PROGRAM StartStop
VAR
	Start:BOOL;	
	Stop:BOOL;	
    Run:BOOL;
	PulseOUT:BOOL;
	Value:INT;
	TOn:TON;	
	Rtrig:R_TRIG;
	TOn_ET: TIME;
	FAIZ: BOOL;
	FAIZV: INT;
	FAIZValue1 : INT;
	FAIZValue2 : INT;
END_VAR

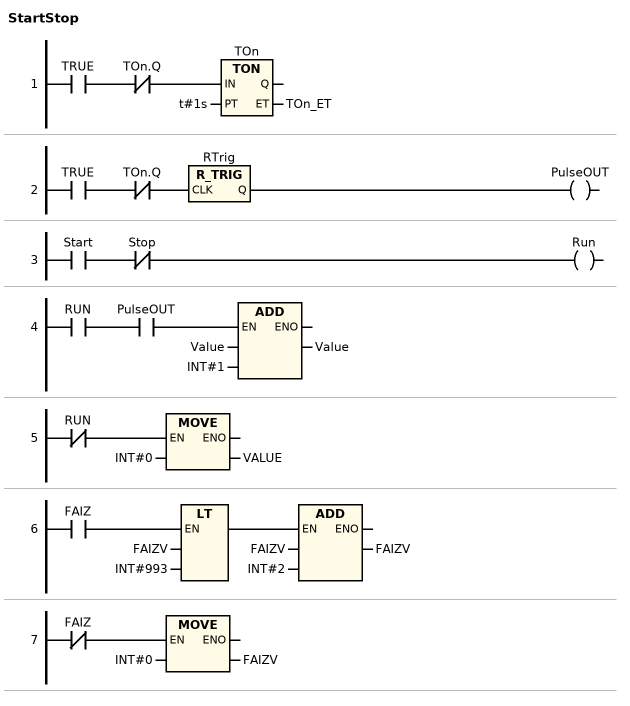
// NETWORK 1
TOn(IN := TRUE AND NOT TOn.Q, PT := t#1s, ET => TOn_ET);

// NETWORK 2
RTrig(CLK := TRUE AND NOT TOn.Q); // R_TRIG
PulseOUT := RTrig.Q;

// NETWORK 3
Run := Start AND NOT Stop;

// NETWORK 4
IF RUN AND PulseOUT THEN Value := Value + INT#1; END_IF

// NETWORK 5
IF NOT RUN THEN VALUE := INT#0; END_IF

// NETWORK 6
IF FAIZ AND FAIZV < INT#993 THEN FAIZV := FAIZV + INT#2; END_IF

// NETWORK 7
IF NOT FAIZ THEN FAIZV := INT#0; END_IF

END_PROGRAM

(* stored: Version 1.1.0.1, ProductVersion 3.1.4024.12
   POU StartStop: Id {0a69edd3-766e-4a2e-bc64-c8e5b893e6c0}, SpecialFunc None *)
